// TIA Portal V20 export
TYPE "zm_Diagnostics"
// stored: Access Published
   STRUCT
      Heartbeat : Bool;
      "CPU Run" : Bool;
   END_STRUCT;
END_TYPE
